{attribute addProperty BoxType "EJ7342-0000-0019"}
{attribute addProperty Id "StatusAT %I*Status_1C57BC2B162"}
{attribute addProperty CRC "3266366177"}
{attribute addProperty SizeInBites "16"}
{attribute addProperty SizeInBytes "2"}
TYPE DCM_Status_Channel_C2B0CAE1 :
STRUCT
	{attribute addProperty Name "Status"}
	Status AT %I* : Status_1C57BC2B;
END_STRUCT
END_TYPE

(* stored: Version 1.2.0.0, ProductVersion 3.1.4024.9
   DUT DCM_Status_Channel_C2B0CAE1: Id {438cc16d-b459-4b41-ba87-df3664f6e693} *)
